# EPICS substitutions: db/Beckhoff_3XXX/ecmcEL3204.substitutions
file "ecmcEcSlave.template"
{
  pattern {}
          {}
}

file "ecmc_analogInput-chX.template"
{
  pattern {CH_ID, ESLO, EOFF, EGU,     PREC}
          {01,     0.1,  0,    "DegC", 2   }
          {02,     0.1,  0,    "DegC", 2   }
          {03,     0.1,  0,    "DegC", 2   }
          {04,     0.1,  0,    "DegC", 2   }
}

file "ecmc_status-chX.template"
{
  pattern {CH_ID, KEY }
          {01,    "AI"}
          {02,    "AI"}
          {03,    "AI"}
          {04,    "AI"}
}
